Omron CX-Programmer project NewProject (CX-Programmer 9.61)

# PLC NewPLC1: CJ2M CPU11
I/O table (CPU CJ2M-CPU11): rack 0 slot 0 CJ1W-ID211; rack 0 slot 1 CJ1W-OD211; rack 0 slot 2 CJ1W-ID211; rack 0 slot 3 CJ1W-OD211; rack 0 slot 4 CJ1W-ID211

## Global symbols (name address type ; comment)
0.00 BOOL  ; EMERGENCY BUTTON
0.01 BOOL  ; SENSOR PRESS UP END(BELUM ADA)
0.02 BOOL  ; PB RESET
0.04 BOOL  ; PX CLAMP
0.05 BOOL  ; SENSOR W/P LASER CONF
0.06 BOOL  ; YELLOW BOX
0.07 BOOL  ; CY FWD LOCK PRESS
0.08 BOOL  ; CY BKWD UNLOCK PRESS
0.09 BOOL  ; SENSOR PRESS DOWN END
0.10 BOOL  ; SENSOR COLOR
0.11 BOOL  ; SENSOR STOPPER RELEASE
0.12 BOOL  ; PIGTAIL CHECK 1
0.13 BOOL  ; PIGTAIL CHECK 2
0.14 BOOL  ; AS FWD STOPPER 2
0.15 BOOL  ; AS BWD STOPPER 2
100.00 BOOL  ; HOME POS
100.01 BOOL  ; STEP1
100.02 BOOL  ; STEP2
100.03 BOOL  ; STEP3
100.04 BOOL  ; AMBIL WORKP
100.05 BOOL  ; CLAIMP OK/NG D92A
100.06 BOOL  ; HOLD SAFETY LIGHT D92A
101.00 BOOL  ; CLAMP W/P
101.01 BOOL  ; YELLOW BOX
101.05 BOOL  ; SALAH MODEL D55L
101.06 BOOL  ; HOLD SAFETY HOLD D55L
111.00 BOOL  ; PUT YELLOW BOX
111.01 BOOL  ; RESET
111.02 BOOL  ; CYD STOPPER FWD AFTER ALARM
1.00 BOOL  ; PL GOOD
1.01 BOOL  ; PL NG
1.02 BOOL  ; SOL CY FWD LOCK PRESS
1.03 BOOL  ; SOL CY BKWD UNLOCK PRESS
1.04 BOOL  ; SOL STOPPER 1
1.05 BOOL  ; BUZZER
1.06 BOOL  ; BUZZER
1.07 BOOL  ; HOME POSITION PL
1.08 BOOL  ; OK PL
1.09 BOOL  ; NG PL
1.10 BOOL  ; AUTO CONDITION PL
1.11 BOOL  ; GREASE COIL CFRM
1.12 BOOL  ; PUNCH UP PL
1.13 BOOL  ; PUNCH DOWN PL
1.14 BOOL  ; TRANSFER FWD PL
1.15 BOOL  ; TRANSFER BWD PL
2000.01 BOOL  ; AUTO START
200.00 BOOL  ; YELLOW BOX
200.01 BOOL  ; AUTO RUNNING
200.02 BOOL  ; AUTO CONDITION
200.03 BOOL  ; TRANSFER START
200.05 BOOL  ; Auto Run Spring Press
200.07 BOOL  ; Slide Door UP each master on
200.08 BOOL  ; GUIDE PALLET BWD EACH MASTERON
200.09 BOOL  ; GUIDE PALLET BWD
20.01 BOOL  ; 1.00
2400.00 BOOL  ; TAKE YELLOW BOX
2400.01 BOOL  ; NG PROSES RESET
2500.01 BOOL  ; STEP PUNCH DOWN
2500.02 BOOL  ; NG PROSES
2500.03 BOOL  ; STEP PUNCH UP
2500.04 BOOL  ; PIGTAIL OK
2500.05 BOOL  ; BEEP OK
2500.06 BOOL  ; NG NO PROSES
2500.07 BOOL  ; FAULT RESET
2500.08 BOOL  ; STOPPER  1 OPEN
2500.09 BOOL  ; READY TRANSFER
2500.10 BOOL  ; Indv WorkPiece Conf
2500.11 BOOL  ; General Error
250.00 BOOL  ; NG NO CAP
250.01 BOOL  ; NG NO PACKING
250.02 BOOL  ; NG NO CAP DAN PACKING
250.03 BOOL  ; skip proses
250.07 BOOL  ; SKIP PROSES D92A
250.08 BOOL  ; NG SKIP PROSES D92A
250.10 BOOL  ; NG SKIP PROSES
251.07 BOOL  ; SKIP PROSES D55L
251.08 BOOL  ; NG SKIP PROSES D55L
2599.00 BOOL  ; Slide door down
2599.01 BOOL  ; Spring Press Down
2599.02 BOOL  ; Cyl Spring Down Comp
2599.03 BOOL  ; Spring Press Up
2599.04 BOOL  ; Spring Press Up Comp
2599.05 BOOL  ; Feeder Pigtail Process
2600.00 BOOL  ; TRANSFER FWD
2600.01 BOOL  ; TRANSFER BWD 1
2600.02 BOOL  ; STOPPER 2 OPEN
2600.03 BOOL  ; TRANSFER BWD 2
2600.04 BOOL  ; TRANSFER BWD 2
2600.06 BOOL  ; Process 1 is Comp
2600.07 BOOL  ; Feeder For Pigtail Process
2600.08 BOOL  ; Holding next process
2600.09 BOOL  ; Next Process after error
2600.10 BOOL  ; Holding next process NG
2600.11 BOOL  ; Slide door up
2600.13 BOOL  ; GUIDE PALLET FORWARD
2.00 BOOL  ; SCREEN
2.01 BOOL  ; CYCLE START
2.02 BOOL  ; SELECT CAP MODEL 2
2.03 BOOL  ; SELECT CAP MODEL 3
2.04 BOOL  ; AS FWD STOPPER 1
2.05 BOOL  ; AS BWD STOPPER 1
2.06 BOOL  ; SENSOR YELLOW BOX
2.07 BOOL  ; PX PALLET1 CFRM
2.09 BOOL  ; PX PALLET2 CFRM
2.10 BOOL  ; AS FWD TRANSFER 2
2.11 BOOL  ; SENSOR CEK CAP
300.00 BOOL  ; FAULT
300.01 BOOL  ; ERROR
300.02 BOOL  ; NO PROSES
300.03 BOOL  ; PALLET 2 DELAY
300.04 BOOL  ; PALLET 1 DELAY
300.06 BOOL  ; Error process
300.07 BOOL  ; Second Process error
300.08 BOOL  ; Process 2nd no detected work/pallet
300.09 BOOL  ; Actuator Error
300.10 BOOL  ; Pallet not going out
300.11 BOOL  ; Machine Overtime Process
300.12 BOOL  ; Feeder When SP Abnormal
300.13 BOOL  ; WORK HAPPENED ERROR
300.14 BOOL  ; Pallet Error
300.15 BOOL  ; 2ND Still Process
301.00 BOOL  ; SP Abnormal slide up
301.01 BOOL  ; Slide Door Up
301.02 BOOL  ; Second Process Work Detected error
301.03 BOOL  ; Sol Spring up ( Abnormal Condition)
301.04 BOOL  ; Spring press down overtime ( Abnormal Condition)
30.00 BOOL  ; PUT WORKPIECE NG
350.00 BOOL  ; alarm 1 cycle
3.00 BOOL  ; SOL TRANSFER BWD 2
3.01 BOOL  ; SPARE
3.02 BOOL  ; SPARE
3.03 BOOL  ; SOL Spring Press Up
3.04 BOOL  ; SOL Spring Press Down
3.05 BOOL  ; PL Spring Press Up
3.06 BOOL  ; PL Spring Press Down
3.07 BOOL  ; Abnormal Relay
3.08 BOOL  ; Slide door up
3.09 BOOL  ; RELLAY ALARM SKIP PROSES
3.10 BOOL  ; SOL GUIDE PALLET BWD
3.11 BOOL  ; SPARE
3.12 BOOL  ; SPARE
3.13 BOOL  ; SPARE
3.14 BOOL  ; SPARE
3.15 BOOL  ; SPARE
4100.00 BOOL  ; AUTO MODE
410.00 BOOL  ; AUTO MODE
4200.00 BOOL  ; INDIVIDU MODE
4400.00 BOOL  ; OK CHECK GREASE & PIGTAIL
4500.00 BOOL  ; AUTO READY
4500.01 BOOL  ; PUNCH DOWN
4500.02 BOOL  ; GREASE CONFIRM
4500.03 BOOL  ; PUNCH UP
4500.04 BOOL  ; PIGTAIL CHECK
4500.05 BOOL  ; STEP END
4500.06 BOOL  ; TRANSFER BWD 1 STANBY
4500.08 BOOL  ; NG PIGTAIL NG GRAESE
4500.09 BOOL  ; OK PIGTAIL NG GREASE
4500.10 BOOL  ; NG PIGTAIL NG GRAESE
4500.11 BOOL  ; OK PIGTAIL NG GREASE
4500.12 BOOL  ; PIGTAIL CHECK 1&2 NG
4500.13 BOOL  ; PIGTAIL CHECK 2 NG
4500.14 BOOL  ; PIGTAIL CHECK 1 NG
4500.15 BOOL  ; CHECK PIGTAIL OK
4600.00 BOOL  ; TRANSFER FWD
4600.01 BOOL  ; TRANSFER BWD 1
4600.02 BOOL  ; STEP END
4600.06 BOOL  ; hold 1 cycle
4700.00 BOOL  ; PUNCH DOWN
4700.01 BOOL  ; PUNCH UP
4700.02 BOOL  ; TRANSFER FWD
4700.03 BOOL  ; TRANSFER BWD
4700.04 BOOL  ; PURGE MANUAL
4700.05 BOOL  ; Spring Press Up
4700.06 BOOL  ; GUIDE PALLET FORWARD
4700.08 BOOL  ; Transfer Backward
4700.09 BOOL  ; Transfer Backward grease
4700.10 BOOL  ; Indiv transfer grease apply
4700.11 BOOL  ; Indv Transfer spring press
4700.12 BOOL  ; indiv transfer both not work
4700.13 BOOL  ; Indiv transfer both work
4700.14 BOOL  ; feeder transfer
4701.00 BOOL  ; Spring Press Down
4.00 BOOL  ; LEAK TEST BELUM PROCES
4.01 BOOL  ; PB Spring Press Down
4.02 BOOL  ; Spring Press Up End
4.03 BOOL  ; Spring Press Down End
4.04 BOOL  ; Area Sensor Spring press
4.05 BOOL  ; Ls. Down limit
4.06 BOOL  ; Work detected SP
4.07 BOOL  ; Slide door up end
4.08 BOOL  ; Slide door down end
4.09 BOOL  ; SENSOR CAP
4.10 BOOL  ; RS GUIDE PALLET BWD
C0002 BOOL  ; AMBIL WORKP D92A
C0003 BOOL  ; AMBIL WORKP D55L
H100 CHANNEL  ; AUTO STEP
H100.00 BOOL  ; STEP 0 AUTO READY
H100.01 BOOL  ; STEP 1 PUNCH DOWN
H100.02 BOOL  ; GREASE CONFIRM
H100.03 BOOL  ; STEP 3 PUNCH UP
H100.04 BOOL  ; PIGTAIL CHECK
H100.05 BOOL  ; STEP END
H100.06 BOOL  ; STEP  6 PALLET TRANSFER
H100.07 BOOL  ; STEP 7 PALLET UNTRANSFER
H100.08 BOOL  ; CYCLE END
H10.00 BOOL  ; W/P SET
H10.01 BOOL  ; YELLOW BOX
H20 CHANNEL  ; AUTO
H200 CHANNEL  ; STEP TRANSFER PALLET
H200.00 BOOL  ; STEP 0 TRANSFER FWD
H200.01 BOOL  ; STEP 1 TRANSFER BWD
H200.02 BOOL  ; STEP END
H200.03 BOOL  ; STEP END
H20.00 BOOL  ; STEP1
H20.01 BOOL  ; STEP2
H20.02 BOOL  ; STEP3
H20.03 BOOL  ; STEP4
T0001 BOOL  ; SENSOR W/P LASER CONF
T0002 BOOL  ; STEP1
T0003 BOOL  ; skip
T0004 BOOL  ; STEP3
T0005 BOOL  ; RESET YELLOW BOX
T0006 BOOL  ; Spring Press Process Error
T0009 BOOL  ; WORKPIECE CFRM
T0010 BOOL  ; PALLET CFRM
T0011 BOOL  ; TIMER STOPPER RELEASE
T0012 BOOL  ; TIMER PIGTAIL CHECK 1 OK
T0013 BOOL  ; TIMER PIGTAIL CHECK 2 OK
T0022 BOOL  ; TIMER PIGTAIIL CHECK1 NG
T0023 BOOL  ; TIMER PIGTAIL CHECK2 NG
T0027 BOOL  ; TIMER PALLET OPEN
T0028 BOOL  ; Holding Timing Down
T0030 BOOL  ; TIMER NO GREASE CHECK
T0090 BOOL  ; TIMER NO WORKPIECE
T0099 BOOL  ; TIMER 2  PIGTAIL OK
T0100 BOOL  ; SAFETY LIGHT D92A
T0101 BOOL  ; CEK CAP D92A
T0102 BOOL  ; STANDBY D92A
T0103 BOOL  ; STEP2
T0104 BOOL  ; TIMER PIGTAIL CHECK1&2 NG
T0110 BOOL  ; SAFETY LIGHT D55L
T0111 BOOL  ; CEK CAP D55L
T0112 BOOL  ; STANDBY D55L
T0190 BOOL  ; TIMER ON FAULT AUTO SWITCH
T0192 BOOL  ; Cylinder area spring press error
T0200 BOOL  ; TIMER AUTO READY
T0201 BOOL  ; TIMER PUNCH DOWN
T0202 BOOL  ; GREASE CONFIRM
T0203 BOOL  ; TIMER PUNCH UP
T0204 BOOL  ; TIMER PIGTAIL CHECK COMPLATE
T0207 BOOL  ; TIMER PALLET 1 DELAY
T0209 BOOL  ; TIMER PALLET 2 DELAY
T0210 BOOL  ; Second Process no work/ pallet
T0211 BOOL  ; Punch Up Overtime Error
T0212 BOOL  ; Punch Down Overtime Error
T0213 BOOL  ; Transfer 1 BWD Overtime Error
T0214 BOOL  ; Stopper 2 BWD Overtime Error
T0215 BOOL  ; Stopper 1 BWD Overtime Error
T0216 BOOL  ; Transfer 2 BWD Overtime Error
T0217 BOOL  ; Spring press up Overtime Error
T0218 BOOL  ; Spring press down Overtime Error
T0219 BOOL  ; GUIDE PALLET FWD ERROR
T0220 BOOL  ; GUIDE PALLET BWD ERROR
T0224 BOOL  ; Pallet not arrive out
T0225 BOOL  ; Pallet not arrive out
T0226 BOOL  ; WORK ERROR DETECTED
T0227 BOOL  ; Pallet stuck
T0228 BOOL  ; WORK ERROR
T0229 BOOL  ; WORK ERROR
T0230 BOOL  ; WORK ERROR
T0235 BOOL  ; TIMING BEFORE ABNORMAL SPRING DOWN
T0300 BOOL  ; TIMER TRANSFER FWD
T0301 BOOL  ; TIMER TRANSFER BWD
T0310 BOOL  ; process 1 Comp
T0400 BOOL  ; TIMER PURGE MANUAL OFF
T0405 BOOL  ; Pallet SP confrm
T0406 BOOL  ; Pallet grease confrm
W10.00 BOOL  ; D92A
W10.01 BOOL  ; 560B
W10.03 BOOL  ; D55L

## Program NewProgram1 (cyclic task 0)
Local symbols
P_0_3s BOOL
＃1 UINT_BCD
＃１ UINT_BCD

### Section SELECT_MODEL

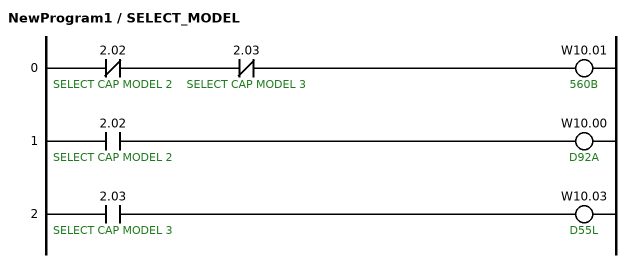
; rung 0
LDNOT 2.02  ; SELECT CAP MODEL 2
ANDNOT 2.03  ; SELECT CAP MODEL 3
OUT W10.01  ; 560B
; rung 1
LD 2.02  ; SELECT CAP MODEL 2
OUT W10.00  ; D92A
; rung 2
LD 2.03  ; SELECT CAP MODEL 3
OUT W10.03  ; D55L

### Section PRESS

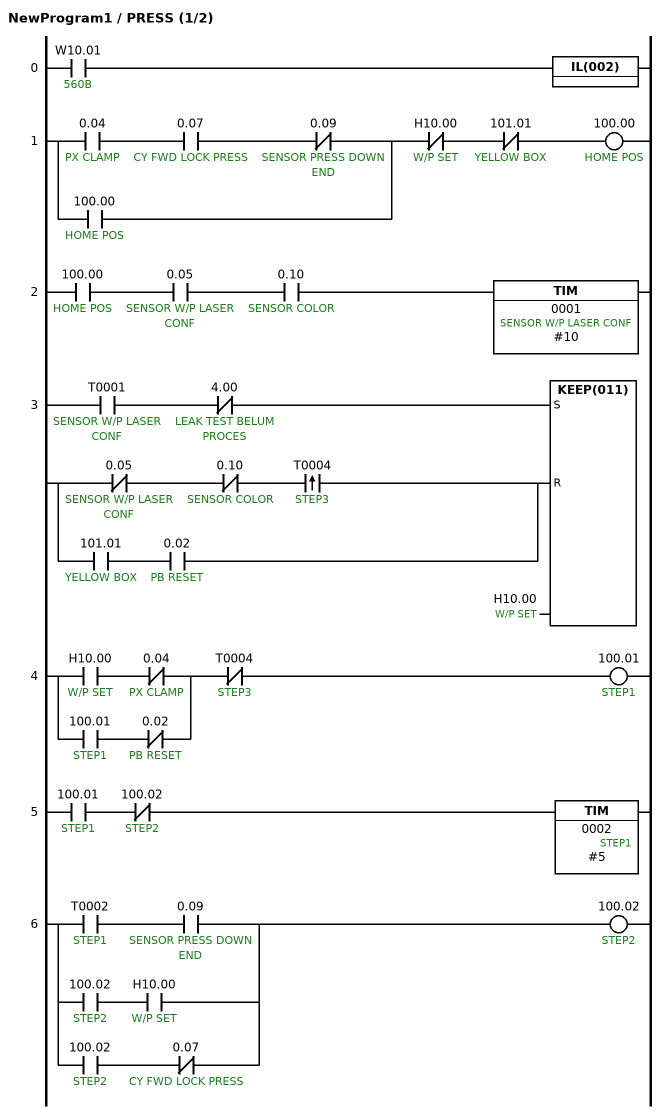
; rung 0
LD W10.01  ; 560B
IL(002)
; rung 1
LD 0.04  ; PX CLAMP
AND 0.07  ; CY FWD LOCK PRESS
ANDNOT 0.09  ; SENSOR PRESS DOWN END
OR 100.00  ; HOME POS
ANDNOT H10.00  ; W/P SET
ANDNOT 101.01  ; YELLOW BOX
OUT 100.00  ; HOME POS
; rung 2
LD 100.00  ; HOME POS
AND 0.05  ; SENSOR W/P LASER CONF
AND 0.10  ; SENSOR COLOR
TIM 0001 #10  ; SENSOR W/P LASER CONF
; rung 3
LD T0001  ; SENSOR W/P LASER CONF
ANDNOT 4.00  ; LEAK TEST BELUM PROCES
LDNOT 0.05  ; SENSOR W/P LASER CONF
ANDNOT 0.10  ; SENSOR COLOR
@AND T0004  ; STEP3
LD 101.01  ; YELLOW BOX
AND 0.02  ; PB RESET
ORLD
KEEP(011) H10.00  ; W/P SET
; rung 4
LD H10.00  ; W/P SET
ANDNOT 0.04  ; PX CLAMP
LD 100.01  ; STEP1
ANDNOT 0.02  ; PB RESET
ORLD
ANDNOT T0004  ; STEP3
OUT 100.01  ; STEP1
; rung 5
LD 100.01  ; STEP1
ANDNOT 100.02  ; STEP2
TIM 0002 #5  ; STEP1
; rung 6
LD T0002  ; STEP1
AND 0.09  ; SENSOR PRESS DOWN END
LD 100.02  ; STEP2
AND H10.00  ; W/P SET
ORLD
LD 100.02  ; STEP2
ANDNOT 0.07  ; CY FWD LOCK PRESS
ORLD
OUT 100.02  ; STEP2

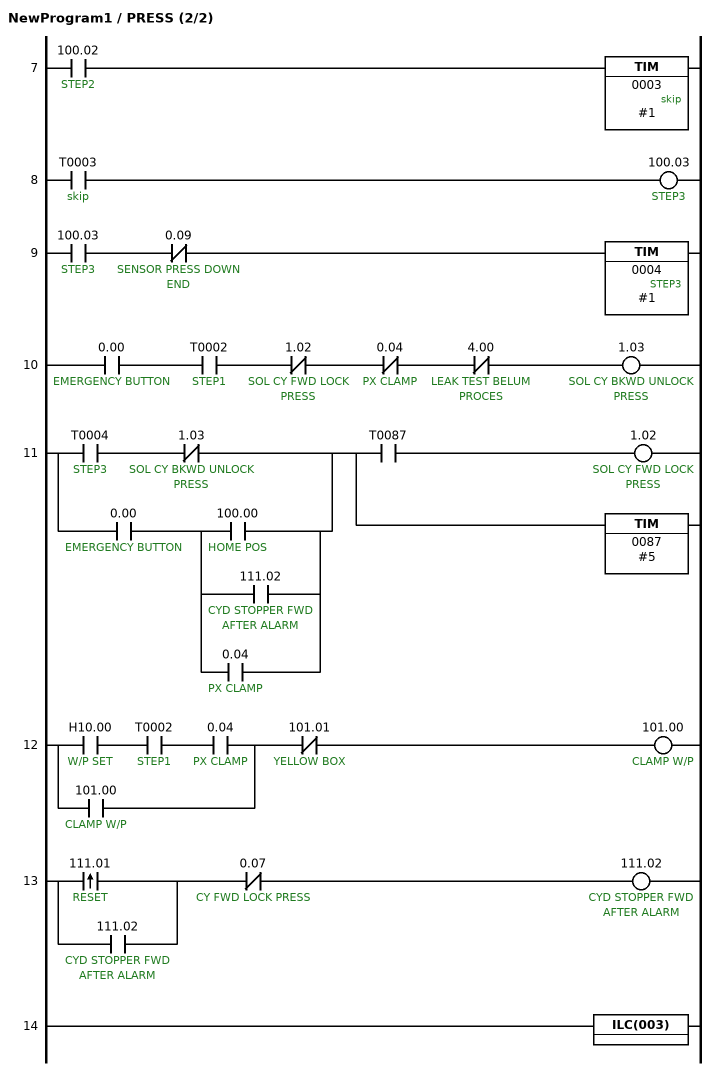
; rung 7
LD 100.02  ; STEP2
TIM 0003 #1  ; skip
; rung 8
LD T0003  ; skip
OUT 100.03  ; STEP3
; rung 9
LD 100.03  ; STEP3
ANDNOT 0.09  ; SENSOR PRESS DOWN END
TIM 0004 #1  ; STEP3
; rung 10
LD 0.00  ; EMERGENCY BUTTON
AND T0002  ; STEP1
ANDNOT 1.02  ; SOL CY FWD LOCK PRESS
ANDNOT 0.04  ; PX CLAMP
ANDNOT 4.00  ; LEAK TEST BELUM PROCES
OUT 1.03  ; SOL CY BKWD UNLOCK PRESS
; rung 11
LD T0004  ; STEP3
ANDNOT 1.03  ; SOL CY BKWD UNLOCK PRESS
LD 0.00  ; EMERGENCY BUTTON
LD 100.00  ; HOME POS
OR 111.02  ; CYD STOPPER FWD AFTER ALARM
OR 0.04  ; PX CLAMP
ANDLD
ORLD
OUT TR0
AND T0087
OUT 1.02  ; SOL CY FWD LOCK PRESS
LD TR0
TIM 0087 #5
; rung 12
LD H10.00  ; W/P SET
AND T0002  ; STEP1
AND 0.04  ; PX CLAMP
OR 101.00  ; CLAMP W/P
ANDNOT 101.01  ; YELLOW BOX
OUT 101.00  ; CLAMP W/P
; rung 13
@LD 111.01  ; RESET
OR 111.02  ; CYD STOPPER FWD AFTER ALARM
ANDNOT 0.07  ; CY FWD LOCK PRESS
OUT 111.02  ; CYD STOPPER FWD AFTER ALARM
; rung 14
ILC(003)

### Section POKAYOKE_CAP_D92A

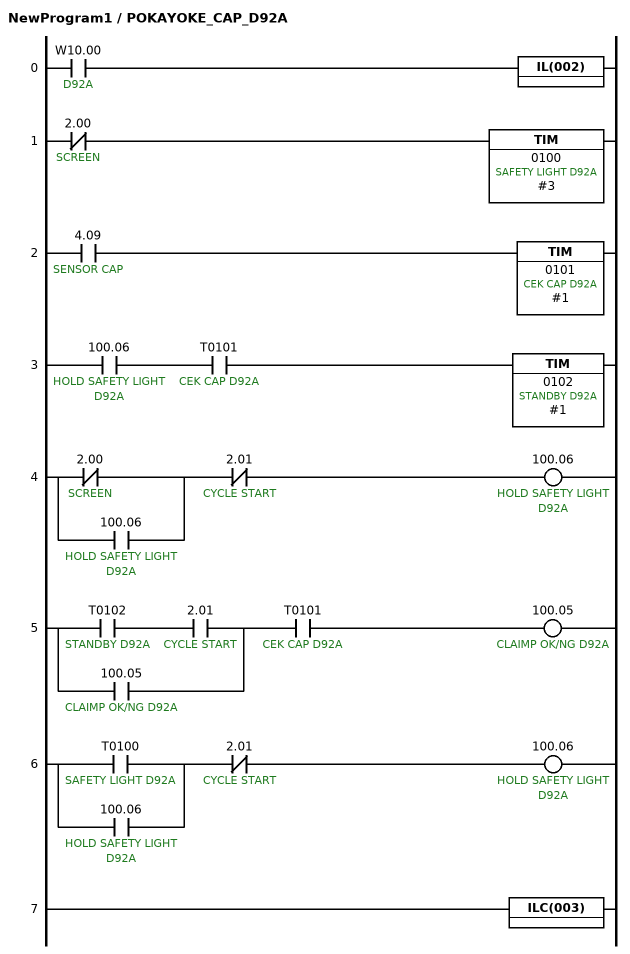
; rung 0
LD W10.00  ; D92A
IL(002)
; rung 1
LDNOT 2.00  ; SCREEN
TIM 0100 #3  ; SAFETY LIGHT D92A
; rung 2
LD 4.09  ; SENSOR CAP
TIM 0101 #1  ; CEK CAP D92A
; rung 3
LD 100.06  ; HOLD SAFETY LIGHT D92A
AND T0101  ; CEK CAP D92A
TIM 0102 #1  ; STANDBY D92A
; rung 4
LDNOT 2.00  ; SCREEN
OR 100.06  ; HOLD SAFETY LIGHT D92A
ANDNOT 2.01  ; CYCLE START
OUT 100.06  ; HOLD SAFETY LIGHT D92A
; rung 5
LD T0102  ; STANDBY D92A
AND 2.01  ; CYCLE START
OR 100.05  ; CLAIMP OK/NG D92A
AND T0101  ; CEK CAP D92A
OUT 100.05  ; CLAIMP OK/NG D92A
; rung 6
LD T0100  ; SAFETY LIGHT D92A
OR 100.06  ; HOLD SAFETY LIGHT D92A
ANDNOT 2.01  ; CYCLE START
OUT 100.06  ; HOLD SAFETY LIGHT D92A
; rung 7
ILC(003)

### Section POKAYOKE_CAP_D55L

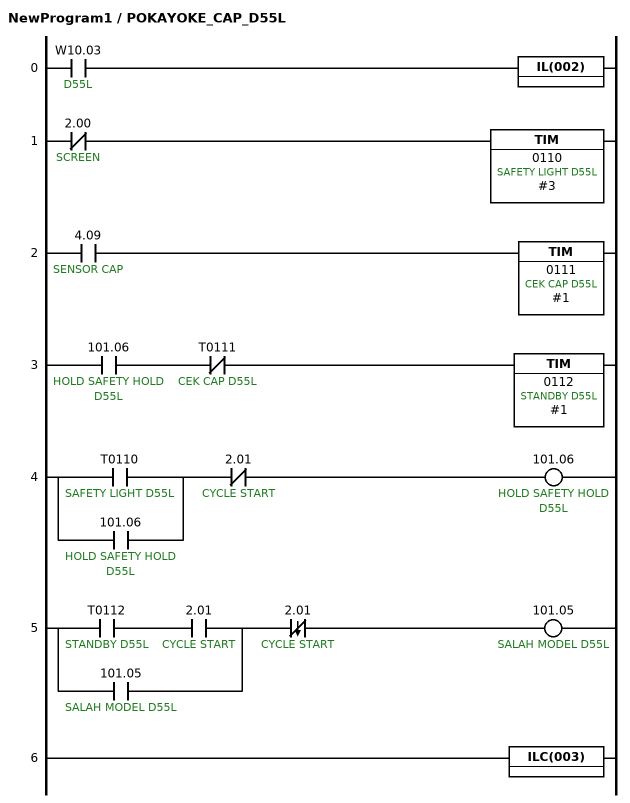
; rung 0
LD W10.03  ; D55L
IL(002)
; rung 1
LDNOT 2.00  ; SCREEN
TIM 0110 #3  ; SAFETY LIGHT D55L
; rung 2
LD 4.09  ; SENSOR CAP
TIM 0111 #1  ; CEK CAP D55L
; rung 3
LD 101.06  ; HOLD SAFETY HOLD D55L
ANDNOT T0111  ; CEK CAP D55L
TIM 0112 #1  ; STANDBY D55L
; rung 4
LD T0110  ; SAFETY LIGHT D55L
OR 101.06  ; HOLD SAFETY HOLD D55L
ANDNOT 2.01  ; CYCLE START
OUT 101.06  ; HOLD SAFETY HOLD D55L
; rung 5
LD T0112  ; STANDBY D55L
AND 2.01  ; CYCLE START
OR 101.05  ; SALAH MODEL D55L
%ANDNOT 2.01  ; CYCLE START
OUT 101.05  ; SALAH MODEL D55L
; rung 6
ILC(003)

### Section FAULT

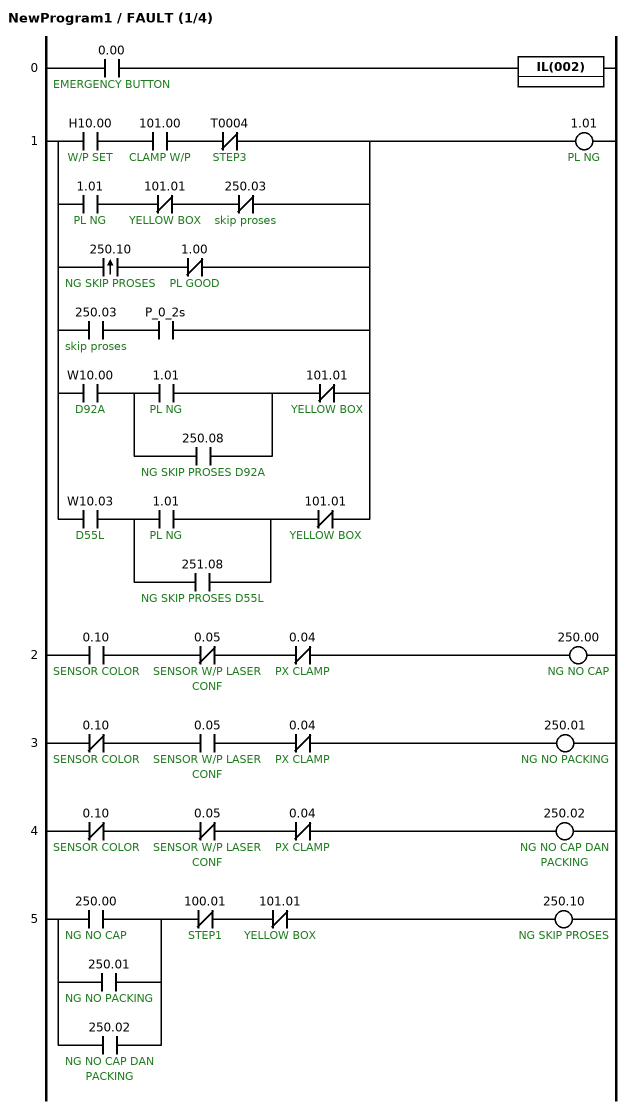
; rung 0
LD 0.00  ; EMERGENCY BUTTON
IL(002)
; rung 1
LD H10.00  ; W/P SET
AND 101.00  ; CLAMP W/P
ANDNOT T0004  ; STEP3
LD 1.01  ; PL NG
ANDNOT 101.01  ; YELLOW BOX
ANDNOT 250.03  ; skip proses
ORLD
@LD 250.10  ; NG SKIP PROSES
ANDNOT 1.00  ; PL GOOD
ORLD
LD 250.03  ; skip proses
AND P_0_2s
ORLD
LD W10.00  ; D92A
LD 1.01  ; PL NG
OR 250.08  ; NG SKIP PROSES D92A
ANDLD
ANDNOT 101.01  ; YELLOW BOX
ORLD
LD W10.03  ; D55L
LD 1.01  ; PL NG
OR 251.08  ; NG SKIP PROSES D55L
ANDLD
ANDNOT 101.01  ; YELLOW BOX
ORLD
OUT 1.01  ; PL NG
; rung 2
LD 0.10  ; SENSOR COLOR
ANDNOT 0.05  ; SENSOR W/P LASER CONF
ANDNOT 0.04  ; PX CLAMP
OUT 250.00  ; NG NO CAP
; rung 3
LDNOT 0.10  ; SENSOR COLOR
AND 0.05  ; SENSOR W/P LASER CONF
ANDNOT 0.04  ; PX CLAMP
OUT 250.01  ; NG NO PACKING
; rung 4
LDNOT 0.10  ; SENSOR COLOR
ANDNOT 0.05  ; SENSOR W/P LASER CONF
ANDNOT 0.04  ; PX CLAMP
OUT 250.02  ; NG NO CAP DAN PACKING
; rung 5
LD 250.00  ; NG NO CAP
OR 250.01  ; NG NO PACKING
OR 250.02  ; NG NO CAP DAN PACKING
ANDNOT 100.01  ; STEP1
ANDNOT 101.01  ; YELLOW BOX
OUT 250.10  ; NG SKIP PROSES

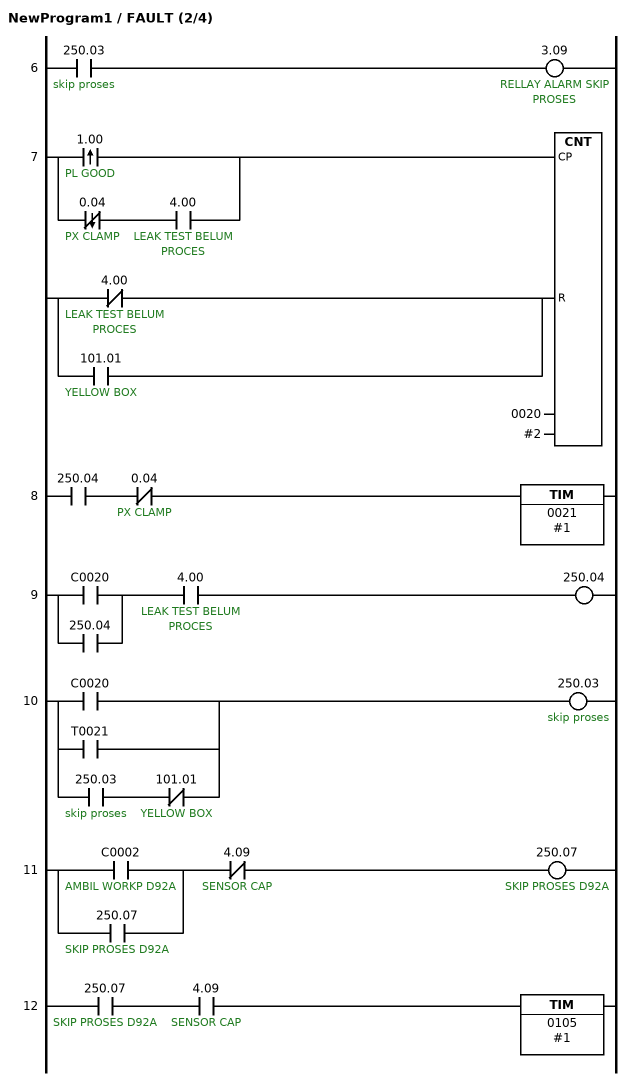
; rung 6
LD 250.03  ; skip proses
OUT 3.09  ; RELLAY ALARM SKIP PROSES
; rung 7
@LD 1.00  ; PL GOOD
%LDNOT 0.04  ; PX CLAMP
AND 4.00  ; LEAK TEST BELUM PROCES
ORLD
LDNOT 4.00  ; LEAK TEST BELUM PROCES
OR 101.01  ; YELLOW BOX
CNT 0020 #2
; rung 8
LD 250.04
ANDNOT 0.04  ; PX CLAMP
TIM 0021 #1
; rung 9
LD C0020
OR 250.04
AND 4.00  ; LEAK TEST BELUM PROCES
OUT 250.04
; rung 10
LD C0020
OR T0021
LD 250.03  ; skip proses
ANDNOT 101.01  ; YELLOW BOX
ORLD
OUT 250.03  ; skip proses
; rung 11
LD C0002  ; AMBIL WORKP D92A
OR 250.07  ; SKIP PROSES D92A
ANDNOT 4.09  ; SENSOR CAP
OUT 250.07  ; SKIP PROSES D92A
; rung 12
LD 250.07  ; SKIP PROSES D92A
AND 4.09  ; SENSOR CAP
TIM 0105 #1

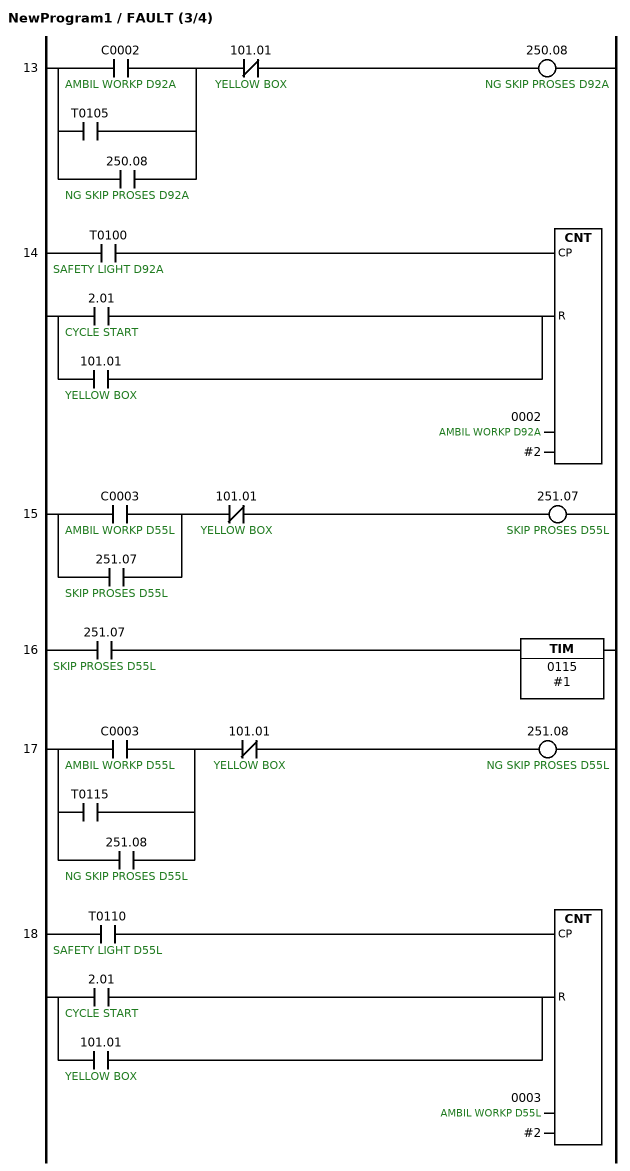
; rung 13
LD C0002  ; AMBIL WORKP D92A
OR T0105
OR 250.08  ; NG SKIP PROSES D92A
ANDNOT 101.01  ; YELLOW BOX
OUT 250.08  ; NG SKIP PROSES D92A
; rung 14
LD T0100  ; SAFETY LIGHT D92A
LD 2.01  ; CYCLE START
OR 101.01  ; YELLOW BOX
CNT 0002 #2  ; AMBIL WORKP D92A
; rung 15
LD C0003  ; AMBIL WORKP D55L
OR 251.07  ; SKIP PROSES D55L
ANDNOT 101.01  ; YELLOW BOX
OUT 251.07  ; SKIP PROSES D55L
; rung 16
LD 251.07  ; SKIP PROSES D55L
TIM 0115 #1
; rung 17
LD C0003  ; AMBIL WORKP D55L
OR T0115
OR 251.08  ; NG SKIP PROSES D55L
ANDNOT 101.01  ; YELLOW BOX
OUT 251.08  ; NG SKIP PROSES D55L
; rung 18
LD T0110  ; SAFETY LIGHT D55L
LD 2.01  ; CYCLE START
OR 101.01  ; YELLOW BOX
CNT 0003 #2  ; AMBIL WORKP D55L

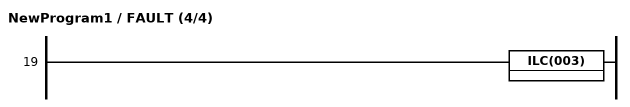
; rung 19
ILC(003)

### Section OUTPUT

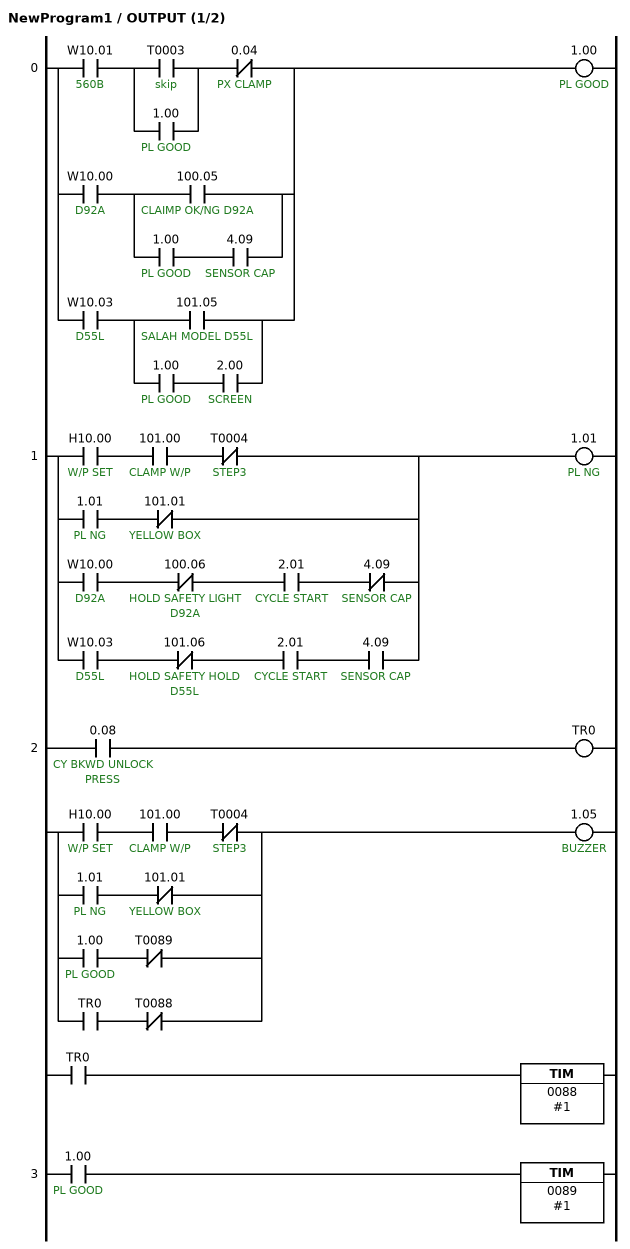
; rung 0
LD W10.01  ; 560B
LD T0003  ; skip
OR 1.00  ; PL GOOD
ANDLD
ANDNOT 0.04  ; PX CLAMP
LD W10.00  ; D92A
LD 100.05  ; CLAIMP OK/NG D92A
LD 1.00  ; PL GOOD
AND 4.09  ; SENSOR CAP
ORLD
ANDLD
ORLD
LD W10.03  ; D55L
LD 101.05  ; SALAH MODEL D55L
LD 1.00  ; PL GOOD
AND 2.00  ; SCREEN
ORLD
ANDLD
ORLD
OUT 1.00  ; PL GOOD
; rung 1
LD H10.00  ; W/P SET
AND 101.00  ; CLAMP W/P
ANDNOT T0004  ; STEP3
LD 1.01  ; PL NG
ANDNOT 101.01  ; YELLOW BOX
ORLD
LD W10.00  ; D92A
ANDNOT 100.06  ; HOLD SAFETY LIGHT D92A
AND 2.01  ; CYCLE START
ANDNOT 4.09  ; SENSOR CAP
ORLD
LD W10.03  ; D55L
ANDNOT 101.06  ; HOLD SAFETY HOLD D55L
AND 2.01  ; CYCLE START
AND 4.09  ; SENSOR CAP
ORLD
OUT 1.01  ; PL NG
; rung 2
LD H10.00  ; W/P SET
AND 101.00  ; CLAMP W/P
ANDNOT T0004  ; STEP3
LD 1.01  ; PL NG
ANDNOT 101.01  ; YELLOW BOX
ORLD
LD 1.00  ; PL GOOD
ANDNOT T0089
ORLD
LD 0.08  ; CY BKWD UNLOCK PRESS
OUT TR0
ANDNOT T0088
ORLD
OUT 1.05  ; BUZZER
LD TR0
TIM 0088 #1
; rung 3
LD 1.00  ; PL GOOD
TIM 0089 #1

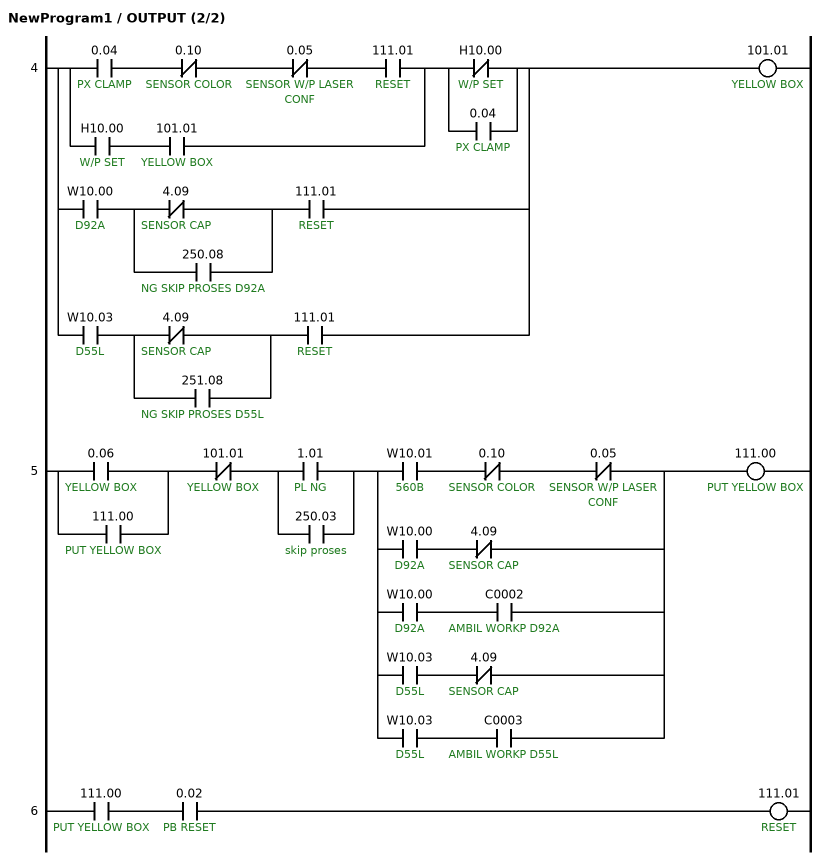
; rung 4
LD 0.04  ; PX CLAMP
ANDNOT 0.10  ; SENSOR COLOR
ANDNOT 0.05  ; SENSOR W/P LASER CONF
AND 111.01  ; RESET
LD H10.00  ; W/P SET
AND 101.01  ; YELLOW BOX
ORLD
LDNOT H10.00  ; W/P SET
OR 0.04  ; PX CLAMP
ANDLD
LD W10.00  ; D92A
LDNOT 4.09  ; SENSOR CAP
OR 250.08  ; NG SKIP PROSES D92A
ANDLD
AND 111.01  ; RESET
ORLD
LD W10.03  ; D55L
LDNOT 4.09  ; SENSOR CAP
OR 251.08  ; NG SKIP PROSES D55L
ANDLD
AND 111.01  ; RESET
ORLD
OUT 101.01  ; YELLOW BOX
; rung 5
LD 0.06  ; YELLOW BOX
OR 111.00  ; PUT YELLOW BOX
ANDNOT 101.01  ; YELLOW BOX
LD 1.01  ; PL NG
OR 250.03  ; skip proses
ANDLD
LD W10.01  ; 560B
ANDNOT 0.10  ; SENSOR COLOR
ANDNOT 0.05  ; SENSOR W/P LASER CONF
LD W10.00  ; D92A
ANDNOT 4.09  ; SENSOR CAP
ORLD
LD W10.00  ; D92A
AND C0002  ; AMBIL WORKP D92A
ORLD
LD W10.03  ; D55L
ANDNOT 4.09  ; SENSOR CAP
ORLD
LD W10.03  ; D55L
AND C0003  ; AMBIL WORKP D55L
ORLD
ANDLD
OUT 111.00  ; PUT YELLOW BOX
; rung 6
LD 111.00  ; PUT YELLOW BOX
AND 0.02  ; PB RESET
OUT 111.01  ; RESET

### Section END
; rung 0
END(001)